FUNCTION_BLOCK CENTRAL_SERVER (* Basic Function Block Type *)
  (* Standard: 61499-2 *)
  (* Version 0.2, 2003-12-04, JHC, Rockwell Automation, Renamed for better indexing. *)
  (* Version 0.1, 2002-11-05, JHC, Rockwell Automation, Corrected missing ST element in Algorithm REQ. *)
  (* Version 0.0, 2000-05-30, JHC, Rockwell Automation *)
  (* Compiler header: package fb.rt.cs725; *)
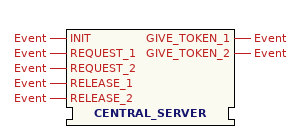
  EVENT_INPUT
    INIT;
    REQUEST_1;
    REQUEST_2;
    RELEASE_1;
    RELEASE_2;
  END_EVENT
  EVENT_OUTPUT
    GIVE_TOKEN_1;
    GIVE_TOKEN_2;
  END_EVENT
  VAR
    requestQueue : ARRAY [0..24] OF INT;
    arrayStartIndex : INT;
    arrayEndIndex : INT;
    tAvailable : BOOL;
    tOwner : INT;
    req1 : BOOL;
    req2 : BOOL;
  END_VAR
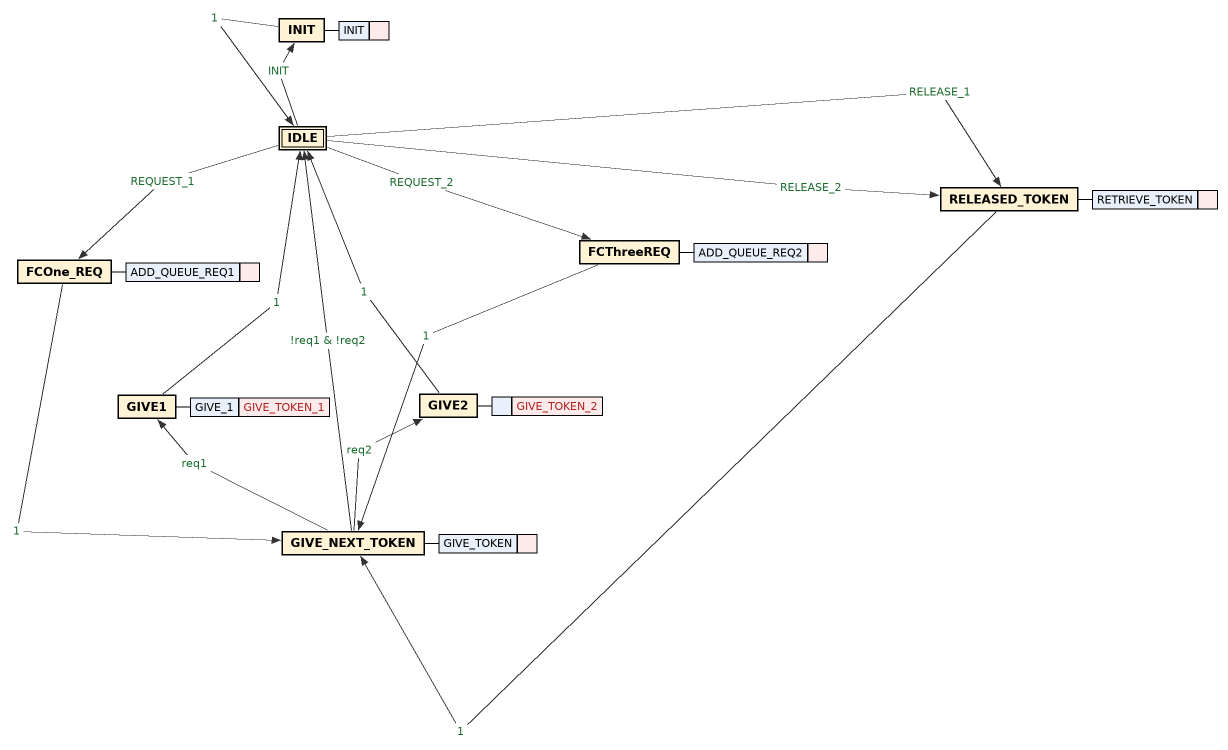
  EC_STATES
    IDLE; (* Initial State *)
    FCOne_REQ : ADD_QUEUE_REQ1;
    FCThreeREQ : ADD_QUEUE_REQ2;
    INIT : INIT;
    GIVE_NEXT_TOKEN : GIVE_TOKEN;
    GIVE2 : -> GIVE_TOKEN_2;
    GIVE1 : GIVE_1 -> GIVE_TOKEN_1;
    RELEASED_TOKEN : RETRIEVE_TOKEN;
  END_STATES
  EC_TRANSITIONS
    IDLE TO FCThreeREQ := REQUEST_2;
    IDLE TO FCOne_REQ := REQUEST_1;
    IDLE TO INIT := INIT;
    INIT TO IDLE := 1;
    FCThreeREQ TO GIVE_NEXT_TOKEN := 1;
    FCOne_REQ TO GIVE_NEXT_TOKEN := 1;
    GIVE_NEXT_TOKEN TO IDLE := !req1 & !req2;
    GIVE_NEXT_TOKEN TO GIVE2 := req2;
    GIVE2 TO IDLE := 1;
    GIVE1 TO IDLE := 1;
    GIVE_NEXT_TOKEN TO GIVE1 := req1;
    IDLE TO RELEASED_TOKEN := RELEASE_1;
    IDLE TO RELEASED_TOKEN := RELEASE_2;
    RELEASED_TOKEN TO GIVE_NEXT_TOKEN := 1;
  END_TRANSITIONS
  ALGORITHM INIT IN ST:
arrayStartIndex := 0;
arrayEndIndex := 0;
tAvailable := TRUE;
tOwner := 0;
  END_ALGORITHM
  ALGORITHM ADD_QUEUE_REQ2 IN ST:
requestQueue[arrayEndIndex] := 2;
arrayEndIndex := ((arrayEndIndex + 1) % 5);
System.out.println("********REQUEST: From Convayer 6********");
  END_ALGORITHM
  ALGORITHM GIVE_1 IN ST:
System.out.println("********GRANT: TOKEN given to Convayer 2********");
  END_ALGORITHM
  ALGORITHM GIVE_2 IN ST:
System.out.println("********GRANT: TOKEN given to Convayer 6********");
  END_ALGORITHM
  ALGORITHM ADD_QUEUE_REQ1 IN ST:
requestQueue[arrayEndIndex] := 1;
arrayEndIndex := ((arrayEndIndex + 1) % 5);
System.out.println("********REQUEST: From Convayer 2********");
  END_ALGORITHM
  ALGORITHM GIVE_TOKEN IN ST:
IF tAvailable = TRUE THEN
    IF requestQueue[arrayStartIndex] <> 0 THEN
        tAvailable := FALSE;
        tOwner := requestQueue[arrayStartIndex];
        requestQueue[arrayStartIndex] := 0;
        arrayStartIndex := ((arrayStartIndex + 1) % 5);
    END_IF;

    IF tOwner = 2 THEN
//System.out.println("*********6 Has Token********");
    req2 := TRUE;
    req1 := FALSE;

    ELSIF tOwner = 1 THEN
//System.out.println("*********2 has Token********");
    req1 := TRUE;
    req2 := FALSE;
    ELSIF tOwner = 0 THEN
    req2 := FALSE;
    req1 := FALSE;
    END_IF;
ELSE
    req2 := FALSE;
    req1 := FALSE;
END_IF;
  END_ALGORITHM
  ALGORITHM RETRIEVE_TOKEN IN ST:
tAvailable := TRUE;
tOwner := 0;
System.out.println("********RELEASED:Server has token********");
  END_ALGORITHM
END_FUNCTION_BLOCK
